(* Permission Group Handlers *)
TYPE ST_SM_PermissionGroups :
STRUCT
    AutoIntlk : ST_PermIntlk_HMI;
    HomePerm : ST_PermIntlk_HMI;
    ProceedPerm : ST_PermIntlk_HMI;
    StartPerm : ST_PermIntlk_HMI;
END_STRUCT
END_TYPE

(* stored: Version 1.1.0.1, ProductVersion 3.1.4024.13
   DUT ST_SM_PermissionGroups: Id {39e2ee62-de6b-4c55-a068-5814939efbf2} *)
